Fanuc KAREL source: KT00247.KL

PROGRAM KT00247
%NOLOCKGROUP
VAR
  Y1: ARRAY[2] OF BYTE
  H2: ARRAY[2] OF SHORT
  OUT: BOOLEAN
BEGIN
  Y1[1] = 2
    H2[1] = 3
  OUT = Y1[1] OR H2[1]
END KT00247
